{attribute 'qualified_only'}
{attribute 'strict'}
TYPE E_XmlError :
(
    Ok := 0,
    ErrorMaxBufferLen := 1,
    ErrorStringLen := 2,
    Error := 3
) BYTE;
END_TYPE

(* stored: Version 1.1.0.1
   DUT E_XmlError: Id {05a4fdda-1086-47b5-ad10-7c2bac568355} *)
